// TIA Portal V20 export
TYPE "LER_typeProcessDataRecord"
// stored: Access Published
   STRUCT
      parentTracecode : Array[0..17] of Char;
      StationID : Array[0..3] of Char;   // Added ASCII characters to account for A/B Ops (i.e. 410A, 410B)
      ProcessPassFail : SInt;   // Summary of all Processes Pass / Fail results 1=pass, 2=fail
   END_STRUCT;
END_TYPE
